SUBAPPLICATION Bool8_TO_logiBUS_QX8 (* 8 generische digitale Ausgaenge (Kanal frei waehlbar), gemeinsam getriggert durch 1 CNF-Event. Generisch fuer jede 8-Bit-Ausgangsgruppe. *)
  (* Standard: 61499-2 *)
  (* Version 1.0, 2026-09-09, Franz Höpfinger, Meisterschulen am Ostbahnhof, Ausgelagert aus Uebung_060_sub_Outputs (dort an TC-SC gebunden) - die 8 Ausgangskanaele waren zuvor fest importierte Output_Q1..Q8, jetzt als VarDeclaration parametrierbar zur Wiederverwendung fuer beliebige 8-Bit-Ausgangsgruppen. *)
  PACKAGE MyLib::sys;
  IMPORT logiBUS::io::DQ::logiBUS_DO;
  IMPORT logiBUS::io::DQ::logiBUS_DO_S;
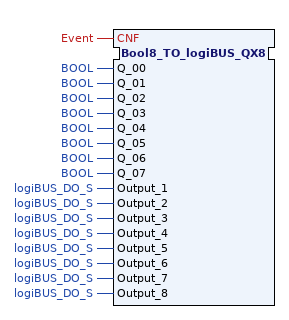
  EVENT_INPUT
    CNF;
  END_EVENT
  VAR_INPUT
    Q_00 : BOOL;
    Q_01 : BOOL;
    Q_02 : BOOL;
    Q_03 : BOOL;
    Q_04 : BOOL;
    Q_05 : BOOL;
    Q_06 : BOOL;
    Q_07 : BOOL;
    Output_1 : logiBUS::io::DQ::logiBUS_DO_S := logiBUS_DO::Invalid; (* Identify the Output Output_Q1..Q8 *)
    Output_2 : logiBUS::io::DQ::logiBUS_DO_S := logiBUS_DO::Invalid; (* Identify the Output Output_Q1..Q8 *)
    Output_3 : logiBUS::io::DQ::logiBUS_DO_S := logiBUS_DO::Invalid; (* Identify the Output Output_Q1..Q8 *)
    Output_4 : logiBUS::io::DQ::logiBUS_DO_S := logiBUS_DO::Invalid; (* Identify the Output Output_Q1..Q8 *)
    Output_5 : logiBUS::io::DQ::logiBUS_DO_S := logiBUS_DO::Invalid; (* Identify the Output Output_Q1..Q8 *)
    Output_6 : logiBUS::io::DQ::logiBUS_DO_S := logiBUS_DO::Invalid; (* Identify the Output Output_Q1..Q8 *)
    Output_7 : logiBUS::io::DQ::logiBUS_DO_S := logiBUS_DO::Invalid; (* Identify the Output Output_Q1..Q8 *)
    Output_8 : logiBUS::io::DQ::logiBUS_DO_S := logiBUS_DO::Invalid; (* Identify the Output Output_Q1..Q8 *)
  END_VAR
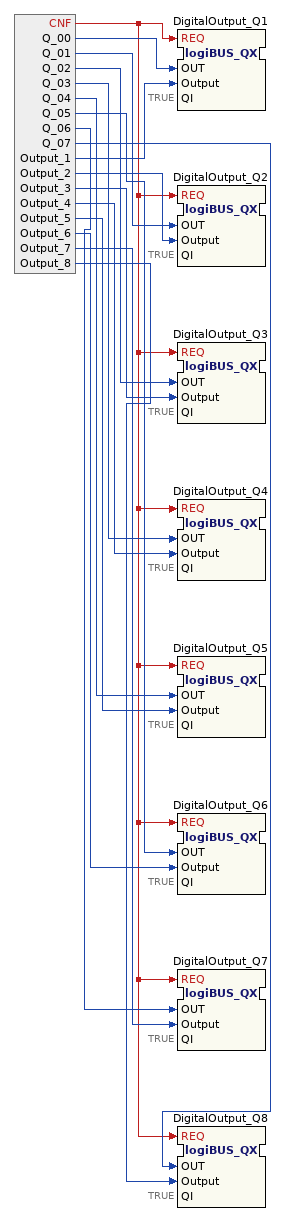
  FBS
    DigitalOutput_Q4 : logiBUS::io::DQ::logiBUS_QX(QI := TRUE);
    DigitalOutput_Q7 : logiBUS::io::DQ::logiBUS_QX(QI := TRUE);
    DigitalOutput_Q1 : logiBUS::io::DQ::logiBUS_QX(QI := TRUE);
    DigitalOutput_Q5 : logiBUS::io::DQ::logiBUS_QX(QI := TRUE);
    DigitalOutput_Q2 : logiBUS::io::DQ::logiBUS_QX(QI := TRUE);
    DigitalOutput_Q6 : logiBUS::io::DQ::logiBUS_QX(QI := TRUE);
    DigitalOutput_Q8 : logiBUS::io::DQ::logiBUS_QX(QI := TRUE);
    DigitalOutput_Q3 : logiBUS::io::DQ::logiBUS_QX(QI := TRUE);
  END_FBS
  EVENT_CONNECTIONS
    CNF TO DigitalOutput_Q4.REQ;
    CNF TO DigitalOutput_Q7.REQ;
    CNF TO DigitalOutput_Q1.REQ;
    CNF TO DigitalOutput_Q5.REQ;
    CNF TO DigitalOutput_Q2.REQ;
    CNF TO DigitalOutput_Q6.REQ;
    CNF TO DigitalOutput_Q8.REQ;
    CNF TO DigitalOutput_Q3.REQ;
  END_CONNECTIONS
  DATA_CONNECTIONS
    Q_06 TO DigitalOutput_Q7.OUT;
    Q_00 TO DigitalOutput_Q1.OUT;
    Q_04 TO DigitalOutput_Q5.OUT;
    Q_01 TO DigitalOutput_Q2.OUT;
    Q_05 TO DigitalOutput_Q6.OUT;
    Q_02 TO DigitalOutput_Q3.OUT;
    Q_03 TO DigitalOutput_Q4.OUT;
    Q_07 TO DigitalOutput_Q8.OUT;
    Output_1 TO DigitalOutput_Q1.Output;
    Output_2 TO DigitalOutput_Q2.Output;
    Output_3 TO DigitalOutput_Q3.Output;
    Output_4 TO DigitalOutput_Q4.Output;
    Output_5 TO DigitalOutput_Q5.Output;
    Output_6 TO DigitalOutput_Q6.Output;
    Output_7 TO DigitalOutput_Q7.Output;
    Output_8 TO DigitalOutput_Q8.Output;
  END_CONNECTIONS
END_SUBAPPLICATION
